// TIA Portal V16 export
// export: Created 2022-07-21T09:35:28.5541146Z, ExportSetting WithDefaults, DisplayName Totally Integrated Automation Portal, DisplayVersion V16 Update 4, DisplayName TIA Portal Version Control Interface, DisplayVersion V16 Update 2, DisplayName TIA Portal Openness, DisplayVersion V16 Update 4, DisplayName SINAMICS Startdrive Advanced, DisplayVersion V16 Update 5, DisplayName SINAMICS Startdrive G130, G150, S120, S150, SINAMICS MV, S210, DisplayVersion V16 Update 5, DisplayName SINAMICS Startdrive G110M, G120, G120C, G120D, G120P, G115D, DisplayVersion V16 Update 5, DisplayName STEP 7 Professional, DisplayVersion V16 Update 4, DisplayName STEP 7 Safety, DisplayVersion V16, DisplayName WinCC Advanced, DisplayVersion V16 Update 4
FUNCTION_BLOCK "fbDriveSiemensSynchro"   // FB707, LAD
TITLE = Drive Siemens Synchro / Drive Siemens jazda synchro
{ S7_Optimized_Access := 'TRUE' }
VERSION : 0.1
// stored: AutoNumber false, IsIECCheckEnabled false, IsRetainMemResEnabled false, MemoryReserve 100, SetENOAutomatically false, UDAEnableTagReadback false
   VAR_INPUT
      executeAbsolute : Bool;
      executeSynchro : Bool;
      stop : Bool;
      extAlm : Bool;
      velocityAuto : LReal;   // [mm/s]
      velocityMan : LReal;   // [mm/s]
      acceleration : LReal;   // [mm/s²]
      decceleration : LReal;   // [mm/s²]
      group : "typeGroup";
      axis : TO_SynchronousAxis;
      master : TO_Axis;
   END_VAR
   VAR_IN_OUT
      drive : "typeDrive";
      axisBasicsDataBlock : "LAxisBasics_typeAxisBasicsData";
      axisConfiguration : "LAxisCtrl_typeAxisConfig";
   END_VAR
   VAR
      delayPTAlm0 : Time := T#1s;   // Czas opóźnienia dla alarmu 0 / alarm delay 0
      delayPTAlm1 : Time := T#1s;   // Czas opóźnienia dla alarmu 1 / alarm delay 1
      delayPTAlm2 : Time := T#1s;   // Czas opóźnienia dla alarmu 2 / alarm delay 2
      delayPTAlm3 : Time := T#1s;   // Czas opóźnienia dla alarmu 3 / alarm delay 3
      delayPTAlm4 : Time := T#1s;   // Czas opóźnienia dla alarmu 4 / alarm delay 4
      delayPTAlm5 : Time := T#1s;   // Czas opóźnienia dla alarmu 5 / alarm delay 5
      delayPTAlm6 : Time := T#1s;   // Czas opóźnienia dla alarmu 6 / alarm delay 6
      delayPTAlm7 : Time := T#1s;   // Czas opóźnienia dla alarmu 7 / alarm delay 7
      instTmrDlyAlm0 { S7_SetPoint := 'True'} : TON_TIME;   // Opóźnienie dla alarmu 0 / alarm delay 0
      instTmrDlyAlm1 { S7_SetPoint := 'True'} : TON_TIME;   // Opóźnienie dla alarmu 1 / alarm delay 1
      instTmrDlyAlm2 { S7_SetPoint := 'True'} : TON_TIME;   // Opóźnienie dla alarmu 2 / alarm delay 2
      instTmrDlyAlm3 { S7_SetPoint := 'True'} : TON_TIME;   // Opóźnienie dla alarmu 3 / alarm delay 3
      instTmrDlyAlm4 { S7_SetPoint := 'True'} : TON_TIME;   // Opóźnienie dla alarmu 4 / alarm delay 4
      instTmrDlyAlm5 { S7_SetPoint := 'True'} : TON_TIME;   // Opóźnienie dla alarmu 5 / alarm delay 5
      instTmrDlyAlm6 { S7_SetPoint := 'True'} : TON_TIME;   // Opóźnienie dla alarmu 6 / alarm delay 6
      instTmrDlyAlm7 { S7_SetPoint := 'True'} : TON_TIME;   // Opóźnienie dla alarmu 7 / alarm delay 7
      instLAxisCtrl_SyncAxisRelGearing { S7_SetPoint := 'True'} : "LAxisCtrl_SyncAxisRelGearing";
      instSetpointVelocity { S7_SetPoint := 'True'} : "fbSPEntryLReal";
      instSetpointPosition { S7_SetPoint := 'True'} : "fbSPEntryLReal";
      statOldAuto { S7_SetPoint := 'True'} : Bool;
      statOldMan : Bool;
      homePulse { S7_SetPoint := 'True'} : TP_TIME;
      DrivecmdExecuteSynchro { S7_SetPoint := 'True'} : Bool;
   END_VAR
   VAR_TEMP
      bAlm0 : Bool;   // tymczasowy bit dla alarmu 0 / temporary alarm bit 0
      bAlm1 : Bool;   // tymczasowy bit dla alarmu 1 / temporary alarm bit 1
      bAlm2 : Bool;   // tymczasowy bit dla alarmu 2 / temporary alarm bit 2
      bAlm3 : Bool;   // tymczasowy bit dla alarmu 3 / temporary alarm bit 3
      bAlm4 : Bool;   // tymczasowy bit dla alarmu 4 / temporary alarm bit 4
      bAlm5 : Bool;   // tymczasowy bit dla alarmu 5 / temporary alarm bit 5
      bAlm6 : Bool;   // tymczasowy bit dla alarmu 6 / temporary alarm bit 6
      bAlm7 : Bool;   // tymczasowy bit dla alarmu 7 / temporary alarm bit 7
      seqStart : Bool;
      "robot in cv zone" : Bool;
   END_VAR
   VAR CONSTANT
      VEL_AUTO : LReal := 500.0;   // prędkość w trybie automatycznym / speed in automatic mode
      VEL_MAN : LReal := 33.0;
      MAX_VEL_AUTO : LReal := 1000.0;   // prędkość w trybie automatycznym / speed in automatic mode
      MAX_VEL_MAN : LReal := 1000.0;
      MIN_VEL : LReal := 0.1;
      MIN_DIST : LReal := 0.0;
      MAX_DIST : LReal := 1232.0;
   END_VAR
   VAR_TEMP   // added for the SCL form of the ladder/FBD networks
      _w1 : Bool;
      _w2 : Bool;
      _w3 : Bool;
   END_VAR
BEGIN

REGION Network 1: Alarm: axis error / Alarm: błąd osi
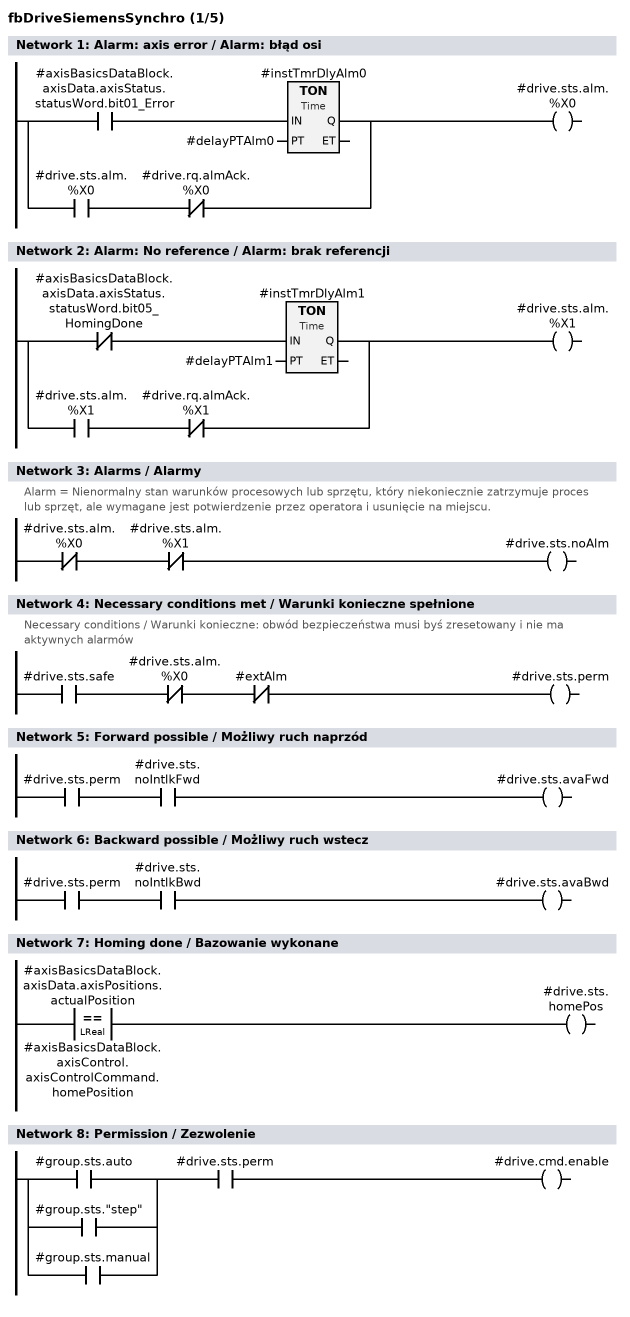
   RUNG wire#powerrail
      Contact( #axisBasicsDataBlock.axisData.axisStatus.statusWord.bit01_Error )
      { S7_Templates := "time_type := Time" } #instTmrDlyAlm0.TON(pt := #delayPTAlm0, et =>)
      wire#w1
      Coil( #drive.sts.alm.%X0 )
   END_RUNG
   RUNG wire#powerrail
      Contact( #drive.sts.alm.%X0 )
      I_Contact( #drive.rq.almAck.%X0 )
   END_RUNG wire#w1
   // the same network as SCL:
   #instTmrDlyAlm0(IN := #axisBasicsDataBlock.axisData.axisStatus.statusWord.bit01_Error, PT := #delayPTAlm0);   // TON
   #drive.sts.alm.%X0 := #instTmrDlyAlm0.Q OR (#drive.sts.alm.%X0 AND NOT #drive.rq.almAck.%X0);
END_REGION

REGION Network 2: Alarm: No reference / Alarm: brak referencji
   RUNG wire#powerrail
      I_Contact( #axisBasicsDataBlock.axisData.axisStatus.statusWord.bit05_HomingDone )
      { S7_Templates := "time_type := Time" } #instTmrDlyAlm1.TON(pt := #delayPTAlm1, et =>)
      wire#w1
      Coil( #drive.sts.alm.%X1 )
   END_RUNG
   RUNG wire#powerrail
      Contact( #drive.sts.alm.%X1 )
      I_Contact( #drive.rq.almAck.%X1 )
   END_RUNG wire#w1
   // the same network as SCL:
   #instTmrDlyAlm1(IN := NOT #axisBasicsDataBlock.axisData.axisStatus.statusWord.bit05_HomingDone,   // TON
                   PT := #delayPTAlm1);
   #drive.sts.alm.%X1 := #instTmrDlyAlm1.Q OR (#drive.sts.alm.%X1 AND NOT #drive.rq.almAck.%X1);
END_REGION

REGION Network 3: Alarms / Alarmy
   // Alarm = Nienormalny stan warunków procesowych lub sprzętu, który niekoniecznie zatrzymuje proces lub sprzęt, ale wymagane jest potwierdzenie przez operatora i usunięcie na miejscu.
   RUNG wire#powerrail
      I_Contact( #drive.sts.alm.%X0 )
      I_Contact( #drive.sts.alm.%X1 )
      Coil( #drive.sts.noAlm )
   END_RUNG
   // the same network as SCL:
   #drive.sts.noAlm := NOT #drive.sts.alm.%X0 AND NOT #drive.sts.alm.%X1;
END_REGION

REGION Network 4: Necessary conditions met / Warunki konieczne spełnione
   // Necessary conditions / Warunki konieczne: obwód bezpieczeństwa musi byś zresetowany i nie ma aktywnych alarmów
   RUNG wire#powerrail
      Contact( #drive.sts.safe )
      I_Contact( #drive.sts.alm.%X0 )
      I_Contact( #extAlm )
      Coil( #drive.sts.perm )
   END_RUNG
   // the same network as SCL:
   #drive.sts.perm := #drive.sts.safe AND NOT #drive.sts.alm.%X0 AND NOT #extAlm;
END_REGION

REGION Network 5: Forward possible / Możliwy ruch naprzód
   RUNG wire#powerrail
      Contact( #drive.sts.perm )
      Contact( #drive.sts.noIntlkFwd )
      Coil( #drive.sts.avaFwd )
   END_RUNG
   // the same network as SCL:
   #drive.sts.avaFwd := #drive.sts.perm AND #drive.sts.noIntlkFwd;
END_REGION

REGION Network 6: Backward possible / Możliwy ruch wstecz
   RUNG wire#powerrail
      Contact( #drive.sts.perm )
      Contact( #drive.sts.noIntlkBwd )
      Coil( #drive.sts.avaBwd )
   END_RUNG
   // the same network as SCL:
   #drive.sts.avaBwd := #drive.sts.perm AND #drive.sts.noIntlkBwd;
END_REGION

REGION Network 7: Homing done / Bazowanie wykonane
   RUNG wire#powerrail
      { S7_Templates := "SrcType := LReal" } EQ_Contact(in1 := #axisBasicsDataBlock.axisData.axisPositions.actualPosition, in2 := #axisBasicsDataBlock.axisControl.axisControlCommand.homePosition)
      Coil( #drive.sts.homePos )
   END_RUNG
   // the same network as SCL:
   #drive.sts.homePos := #axisBasicsDataBlock.axisData.axisPositions.actualPosition = #axisBasicsDataBlock.axisControl.axisControlCommand.homePosition;
END_REGION

REGION Network 8: Permission / Zezwolenie
   RUNG wire#powerrail
      Contact( #group.sts.auto )
      wire#w1
      Contact( #drive.sts.perm )
      Coil( #drive.cmd.enable )
   END_RUNG
   RUNG wire#powerrail
      Contact( #group.sts."step" )
   END_RUNG wire#w1
   RUNG wire#powerrail
      Contact( #group.sts.manual )
   END_RUNG wire#w1
   // the same network as SCL:
   #drive.cmd.enable := (#group.sts.auto OR #group.sts."step" OR #group.sts.manual) AND #drive.sts.perm;
END_REGION

REGION Network 9: Forward / W przód
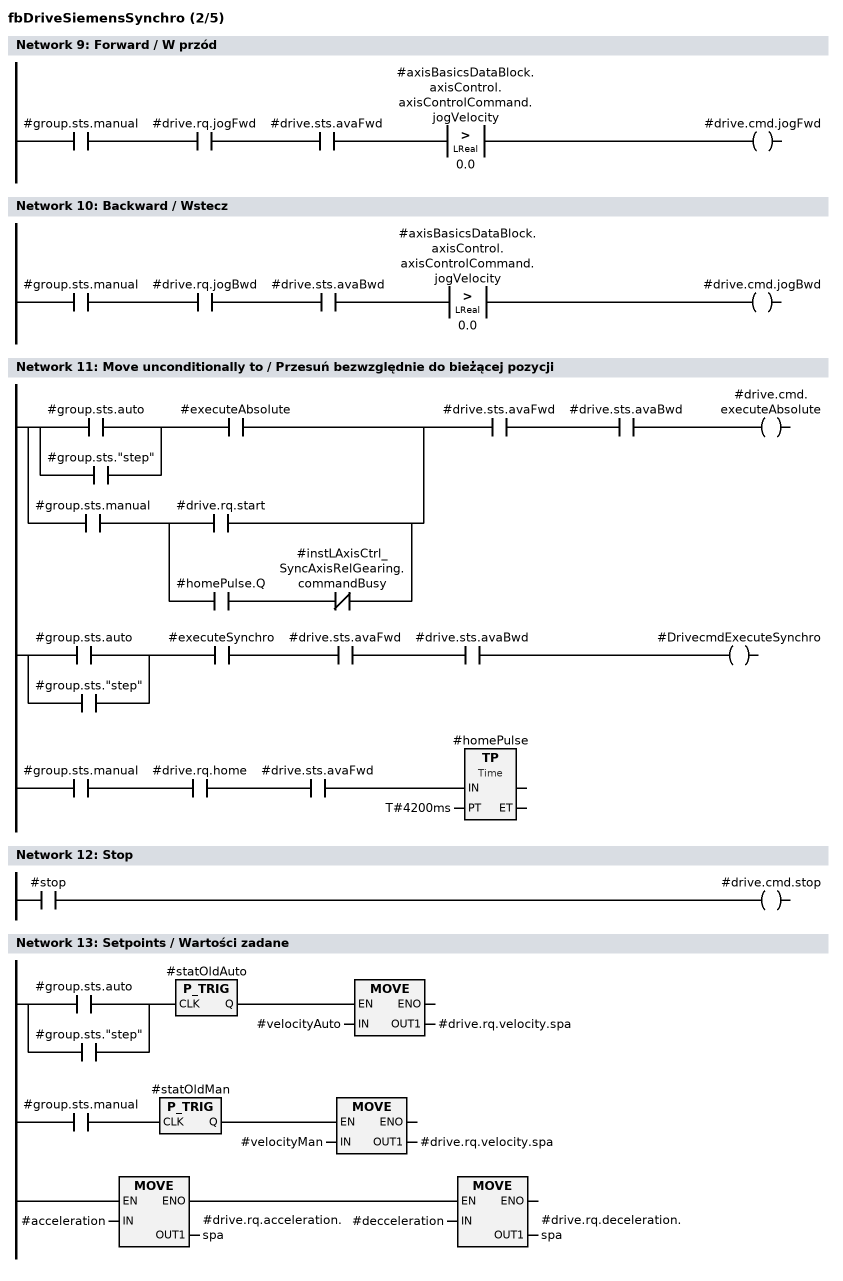
   RUNG wire#powerrail
      Contact( #group.sts.manual )
      Contact( #drive.rq.jogFwd )
      Contact( #drive.sts.avaFwd )
      { S7_Templates := "SrcType := LReal" } GT_Contact(in1 := #axisBasicsDataBlock.axisControl.axisControlCommand.jogVelocity, in2 := 0.0)
      Coil( #drive.cmd.jogFwd )
   END_RUNG
   // the same network as SCL:
   #drive.cmd.jogFwd := #group.sts.manual AND #drive.rq.jogFwd AND #drive.sts.avaFwd AND (#axisBasicsDataBlock.axisControl.axisControlCommand.jogVelocity > 0.0);
END_REGION

REGION Network 10: Backward / Wstecz
   RUNG wire#powerrail
      Contact( #group.sts.manual )
      Contact( #drive.rq.jogBwd )
      Contact( #drive.sts.avaBwd )
      { S7_Templates := "SrcType := LReal" } GT_Contact(in1 := #axisBasicsDataBlock.axisControl.axisControlCommand.jogVelocity, in2 := 0.0)
      Coil( #drive.cmd.jogBwd )
   END_RUNG
   // the same network as SCL:
   #drive.cmd.jogBwd := #group.sts.manual AND #drive.rq.jogBwd AND #drive.sts.avaBwd AND (#axisBasicsDataBlock.axisControl.axisControlCommand.jogVelocity > 0.0);
END_REGION

REGION Network 11: Move unconditionally to / Przesuń bezwzględnie do bieżącej pozycji
   RUNG wire#powerrail
      Contact( #group.sts.auto )
      wire#w1
      Contact( #executeAbsolute )
      wire#w2
      Contact( #drive.sts.avaFwd )
      Contact( #drive.sts.avaBwd )
      Coil( #drive.cmd.executeAbsolute )
   END_RUNG
   RUNG wire#powerrail
      Contact( #group.sts."step" )
   END_RUNG wire#w1
   RUNG wire#powerrail
      Contact( #group.sts.manual )
      wire#w3
      Contact( #drive.rq.start )
   END_RUNG wire#w2
   RUNG wire#w3
      Contact( #homePulse.Q )
      I_Contact( #instLAxisCtrl_SyncAxisRelGearing.commandBusy )
   END_RUNG wire#w2
   RUNG wire#powerrail
      Contact( #group.sts.auto )
      wire#w4
      Contact( #executeSynchro )
      Contact( #drive.sts.avaFwd )
      Contact( #drive.sts.avaBwd )
      Coil( #DrivecmdExecuteSynchro )
   END_RUNG
   RUNG wire#powerrail
      Contact( #group.sts."step" )
   END_RUNG wire#w4
   RUNG wire#powerrail
      Contact( #group.sts.manual )
      Contact( #drive.rq.home )
      Contact( #drive.sts.avaFwd )
      { S7_Templates := "time_type := Time" } #homePulse.TP(pt := T#4200ms, et =>)
   END_RUNG
   // the same network as SCL:
   #drive.cmd.executeAbsolute := (((#group.sts.auto OR #group.sts."step") AND #executeAbsolute) OR (#group.sts.manual AND (#drive.rq.start OR (#homePulse.Q AND NOT #instLAxisCtrl_SyncAxisRelGearing.commandBusy)))) AND #drive.sts.avaFwd AND #drive.sts.avaBwd;
   #DrivecmdExecuteSynchro := (#group.sts.auto OR #group.sts."step") AND #executeSynchro AND #drive.sts.avaFwd AND #drive.sts.avaBwd;
   #homePulse(IN := #group.sts.manual AND #drive.rq.home AND #drive.sts.avaFwd, PT := T#4200ms);   // TP
END_REGION

REGION Network 12: Stop
   RUNG wire#powerrail
      Contact( #stop )
      Coil( #drive.cmd.stop )
   END_RUNG
   // the same network as SCL:
   #drive.cmd.stop := #stop;
END_REGION

REGION Network 13: Setpoints / Wartości zadane
   RUNG wire#powerrail
      Contact( #group.sts.auto )
      wire#w1
      P_Trig( #statOldAuto )
      Move(in := #velocityAuto, out1 => #drive.rq.velocity.spa)
   END_RUNG
   RUNG wire#powerrail
      Contact( #group.sts."step" )
   END_RUNG wire#w1
   RUNG wire#powerrail
      Contact( #group.sts.manual )
      P_Trig( #statOldMan )
      Move(in := #velocityMan, out1 => #drive.rq.velocity.spa)
   END_RUNG
   RUNG wire#powerrail
      Move(in := #acceleration, out1 => #drive.rq.acceleration.spa)
      Move(in := #decceleration, out1 => #drive.rq.deceleration.spa)
   END_RUNG
   // the same network as SCL:
   #_w1 := #group.sts.auto OR #group.sts."step";
   #_w2 := #_w1 AND NOT #statOldAuto;   // rising edge
   #statOldAuto := #_w1;
   IF #_w2 THEN #drive.rq.velocity.spa := #velocityAuto; END_IF;
   #_w3 := #group.sts.manual AND NOT #statOldMan;   // rising edge
   #statOldMan := #group.sts.manual;
   IF #_w3 THEN #drive.rq.velocity.spa := #velocityMan; END_IF;
   #drive.rq.acceleration.spa := #acceleration;
   #drive.rq.deceleration.spa := #decceleration;
END_REGION

REGION Network 14: Preset velocity / Prędkość zadana
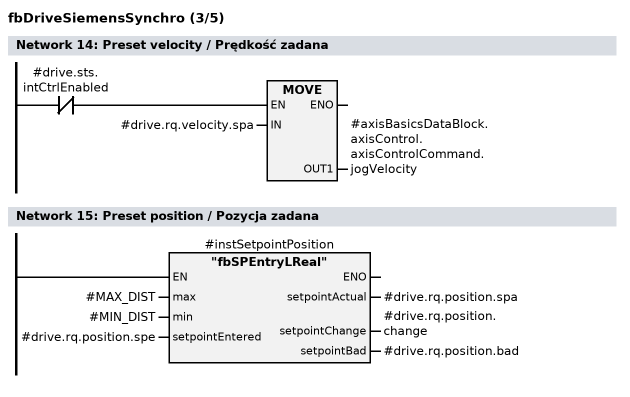
   RUNG wire#powerrail
      I_Contact( #drive.sts.intCtrlEnabled )
      Move(in := #drive.rq.velocity.spa, out1 => #axisBasicsDataBlock.axisControl.axisControlCommand.jogVelocity)
   END_RUNG
   // the same network as SCL:
   IF NOT #drive.sts.intCtrlEnabled THEN
       #axisBasicsDataBlock.axisControl.axisControlCommand.jogVelocity := #drive.rq.velocity.spa;
   END_IF;
END_REGION

REGION Network 15: Preset position / Pozycja zadana
   RUNG wire#powerrail
      #instSetpointPosition(max := #MAX_DIST, min := #MIN_DIST, setpointEntered := #drive.rq.position.spe, setpointActual => #drive.rq.position.spa, setpointChange => #drive.rq.position.change, setpointBad => #drive.rq.position.bad)
   END_RUNG
   // the same network as SCL:
   #instSetpointPosition(max := #MAX_DIST,   // "fbSPEntryLReal"
                         min := #MIN_DIST,
                         setpointEntered := #drive.rq.position.spe,
                         setpointActual => #drive.rq.position.spa,
                         setpointChange => #drive.rq.position.change,
                         setpointBad => #drive.rq.position.bad);
END_REGION

REGION Network 16 (SCL): Copy DB -> Configuration / Przepisanie DB -> Configuration
   //power
   #axisConfiguration.power.startMode := 1;

   //jog mode
   #axisConfiguration.jog.velocity := #axisBasicsDataBlock.axisControl.axisControlCommand.jogVelocity;
   #axisConfiguration.jog.acceleration := #axisBasicsDataBlock.axisControl.axisControlCommand.jogAcceleration;
   #axisConfiguration.jog.deceleration := #axisBasicsDataBlock.axisControl.axisControlCommand.jogDeceleration;
   #axisConfiguration.jog.jerk := #axisBasicsDataBlock.axisControl.axisControlCommand.jogJerk;
   #axisConfiguration.jog.increment := 1;
   #axisConfiguration.jog.positionControlled := #axisBasicsDataBlock.axisControl.axisControlCommand.jogPositionControlled;

   //homing 
   #axisConfiguration.homing.mode := #axisBasicsDataBlock.axisControl.axisControlCommand.homeMode; //7; 
   #axisConfiguration.homing.position := #axisBasicsDataBlock.axisControl.axisControlCommand.homePosition; //0;
   #axisConfiguration.homing.extendedMode := -1; //no extended mode

   //posAbsolute
   #axisConfiguration.posAbsolute.velocity := #drive.rq.velocity.spa;
   #axisConfiguration.posAbsolute.position := #drive.rq.position.spa;
   #axisConfiguration.posAbsolute.acceleration := #drive.rq.acceleration.spa;
   #axisConfiguration.posAbsolute.deceleration := #drive.rq.deceleration.spa;
   #axisConfiguration.posAbsolute.jerk := #axisConfiguration.jog.jerk;
   #axisConfiguration.posAbsolute.direction := 1;

   //synchro
   #axisConfiguration.gearInRelative.ratioNumerator := 1;
   #axisConfiguration.gearInRelative.ratioDenominator := 1;
   #axisConfiguration.gearInRelative.acceleration := #drive.rq.acceleration.spa;
   #axisConfiguration.gearInRelative.deceleration := #drive.rq.deceleration.spa;
   #axisConfiguration.gearInRelative.jerk := #axisConfiguration.jog.jerk;
END_REGION

REGION Network 17: Call: SyncAxisRelGearing / Wywołanie: SyncAxisRelGearing
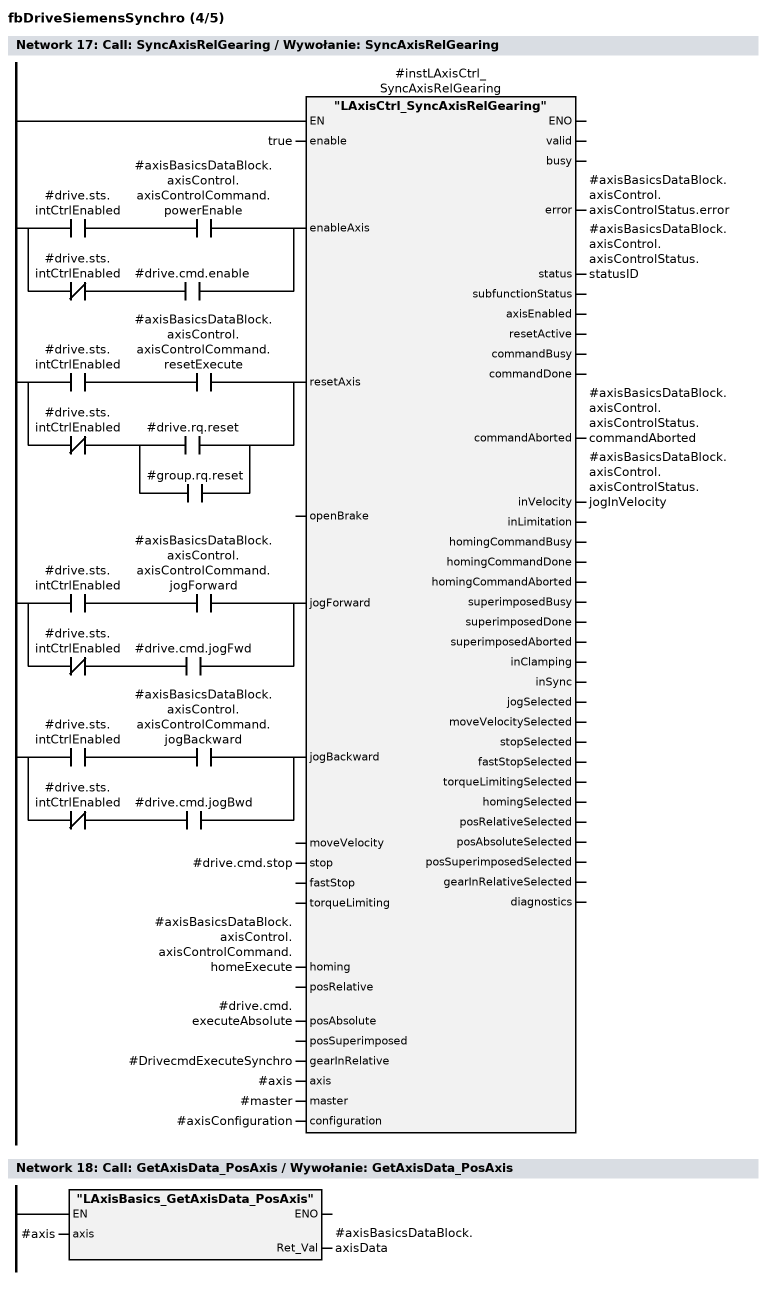
   RUNG wire#powerrail
      #instLAxisCtrl_SyncAxisRelGearing(enableAxis := wire#w1, resetAxis := wire#w3, jogForward := wire#w4, jogBackward := wire#w5, enable := true, openBrake :=, moveVelocity :=, stop := #drive.cmd.stop, fastStop :=, torqueLimiting :=, homing := #axisBasicsDataBlock.axisControl.axisControlCommand.homeExecute, posRelative :=, posAbsolute := #drive.cmd.executeAbsolute, posSuperimposed :=, gearInRelative := #DrivecmdExecuteSynchro, axis := #axis, master := #master, configuration := #axisConfiguration, valid =>, busy =>, error => #axisBasicsDataBlock.axisControl.axisControlStatus.error, status => #axisBasicsDataBlock.axisControl.axisControlStatus.statusID, subfunctionStatus =>, axisEnabled =>, resetActive =>, commandBusy =>, commandDone =>, commandAborted => #axisBasicsDataBlock.axisControl.axisControlStatus.commandAborted, inVelocity => #axisBasicsDataBlock.axisControl.axisControlStatus.jogInVelocity, inLimitation =>, homingCommandBusy =>, homingCommandDone =>, homingCommandAborted =>, superimposedBusy =>, superimposedDone =>, superimposedAborted =>, inClamping =>, inSync =>, jogSelected =>, moveVelocitySelected =>, stopSelected =>, fastStopSelected =>, torqueLimitingSelected =>, homingSelected =>, posRelativeSelected =>, posAbsoluteSelected =>, posSuperimposedSelected =>, gearInRelativeSelected =>, diagnostics =>)
   END_RUNG
   RUNG wire#powerrail
      Contact( #drive.sts.intCtrlEnabled )
      Contact( #axisBasicsDataBlock.axisControl.axisControlCommand.powerEnable )
   END_RUNG wire#w1
   RUNG wire#powerrail
      I_Contact( #drive.sts.intCtrlEnabled )
      Contact( #drive.cmd.enable )
   END_RUNG wire#w1
   RUNG wire#powerrail
      Contact( #drive.sts.intCtrlEnabled )
      Contact( #axisBasicsDataBlock.axisControl.axisControlCommand.resetExecute )
   END_RUNG wire#w3
   RUNG wire#powerrail
      I_Contact( #drive.sts.intCtrlEnabled )
      wire#w2
      Contact( #drive.rq.reset )
   END_RUNG wire#w3
   RUNG wire#w2
      Contact( #group.rq.reset )
   END_RUNG wire#w3
   RUNG wire#powerrail
      Contact( #drive.sts.intCtrlEnabled )
      Contact( #axisBasicsDataBlock.axisControl.axisControlCommand.jogForward )
   END_RUNG wire#w4
   RUNG wire#powerrail
      I_Contact( #drive.sts.intCtrlEnabled )
      Contact( #drive.cmd.jogFwd )
   END_RUNG wire#w4
   RUNG wire#powerrail
      Contact( #drive.sts.intCtrlEnabled )
      Contact( #axisBasicsDataBlock.axisControl.axisControlCommand.jogBackward )
   END_RUNG wire#w5
   RUNG wire#powerrail
      I_Contact( #drive.sts.intCtrlEnabled )
      Contact( #drive.cmd.jogBwd )
   END_RUNG wire#w5
   // the same network as SCL:
   #instLAxisCtrl_SyncAxisRelGearing(enable := true,   // "LAxisCtrl_SyncAxisRelGearing"
                           enableAxis := (#drive.sts.intCtrlEnabled AND #axisBasicsDataBlock.axisControl.axisControlCommand.powerEnable) OR (NOT #drive.sts.intCtrlEnabled AND #drive.cmd.enable),
                           resetAxis := (#drive.sts.intCtrlEnabled AND #axisBasicsDataBlock.axisControl.axisControlCommand.resetExecute) OR (NOT #drive.sts.intCtrlEnabled AND (#drive.rq.reset OR #group.rq.reset)),
                           jogForward := (#drive.sts.intCtrlEnabled AND #axisBasicsDataBlock.axisControl.axisControlCommand.jogForward) OR (NOT #drive.sts.intCtrlEnabled AND #drive.cmd.jogFwd),
                           jogBackward := (#drive.sts.intCtrlEnabled AND #axisBasicsDataBlock.axisControl.axisControlCommand.jogBackward) OR (NOT #drive.sts.intCtrlEnabled AND #drive.cmd.jogBwd),
                           stop := #drive.cmd.stop,
                           homing := #axisBasicsDataBlock.axisControl.axisControlCommand.homeExecute,
                           posAbsolute := #drive.cmd.executeAbsolute,
                           gearInRelative := #DrivecmdExecuteSynchro,
                           axis := #axis,
                           master := #master,
                           configuration := #axisConfiguration,
                           error => #axisBasicsDataBlock.axisControl.axisControlStatus.error,
                           status => #axisBasicsDataBlock.axisControl.axisControlStatus.statusID,
                           commandAborted => #axisBasicsDataBlock.axisControl.axisControlStatus.commandAborted,
                           inVelocity => #axisBasicsDataBlock.axisControl.axisControlStatus.jogInVelocity);
END_REGION

REGION Network 18: Call: GetAxisData_PosAxis / Wywołanie: GetAxisData_PosAxis
   RUNG wire#powerrail
      "LAxisBasics_GetAxisData_PosAxis"(axis := #axis, Ret_Val => #axisBasicsDataBlock.axisData)
   END_RUNG
   // the same network as SCL:
   #axisBasicsDataBlock.axisData := "LAxisBasics_GetAxisData_PosAxis"(axis := #axis);
END_REGION

REGION Network 19 (SCL): Copy LAxisCtrl -> DB / Przepisanie LAxisCtrl -> DB

   #axisBasicsDataBlock.axisControl.axisControlStatus.powerStatus := #instLAxisCtrl_SyncAxisRelGearing.instPower.Status;
   #axisBasicsDataBlock.axisControl.axisControlStatus.powerBusy := #instLAxisCtrl_SyncAxisRelGearing.instPower.Busy;
   #axisBasicsDataBlock.axisControl.axisControlStatus.resetDone := #instLAxisCtrl_SyncAxisRelGearing.instReset.Done;
   #axisBasicsDataBlock.axisControl.axisControlStatus.resetBusy := #instLAxisCtrl_SyncAxisRelGearing.instReset.Busy;

   #axisBasicsDataBlock.axisControl.axisControlStatus.jogBusy := #instLAxisCtrl_SyncAxisRelGearing.instMoveJog.Busy;
   #axisBasicsDataBlock.axisControl.axisControlStatus.homeBusy := #instLAxisCtrl_SyncAxisRelGearing.instHome.Busy;
   #axisBasicsDataBlock.axisControl.axisControlStatus.homeDone := #instLAxisCtrl_SyncAxisRelGearing.instHome.Done;

   #axisBasicsDataBlock.moveToEndPos.moveToEndPosStatus.inPosition := #instLAxisCtrl_SyncAxisRelGearing.instMoveAbsolute.Done;
END_REGION

REGION Network 20: Actual speed / Prędkość rzeczywista
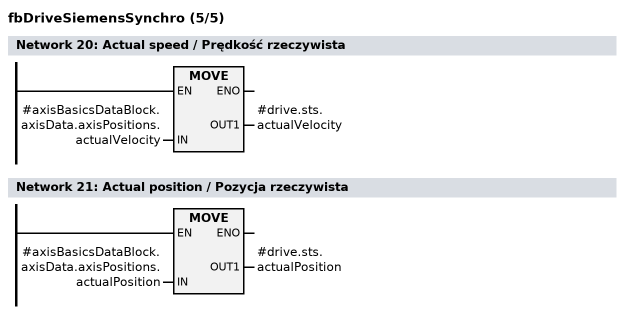
   RUNG wire#powerrail
      Move(in := #axisBasicsDataBlock.axisData.axisPositions.actualVelocity, out1 => #drive.sts.actualVelocity)
   END_RUNG
   // the same network as SCL:
   #drive.sts.actualVelocity := #axisBasicsDataBlock.axisData.axisPositions.actualVelocity;
END_REGION

REGION Network 21: Actual position / Pozycja rzeczywista
   RUNG wire#powerrail
      Move(in := #axisBasicsDataBlock.axisData.axisPositions.actualPosition, out1 => #drive.sts.actualPosition)
   END_RUNG
   // the same network as SCL:
   #drive.sts.actualPosition := #axisBasicsDataBlock.axisData.axisPositions.actualPosition;
END_REGION
END_FUNCTION_BLOCK
